PROGRAM MAIN
VAR
END_VAR

P_Task1();
P_Task2();

END_PROGRAM

(* stored: Version 1.1.0.1, ProductVersion 3.1.4024.12
   POU MAIN: Id {7beae7c3-c9f1-44dc-9799-7da82ef4218c}, SpecialFunc None *)
